PROGRAM MAIN_FAST
VAR
	nCount : INT;
END_VAR

nCount := nCount + 1;
PRG_1();

END_PROGRAM

(* stored: Version 1.1.0.1, ProductVersion 3.1.4024.16
   POU MAIN_FAST: Id {d416186c-e383-4bb0-b869-5e7bc4e524c4}, SpecialFunc None *)
